// TIA Portal project "nalewak_v1" (V20)

(* hardware
DEVICE "S7-1500/ET200MP station_1"  S7-1500 station
   slot 0: "Rail_0"  Rack  6ES7 590-1***0-0AA0
   slot 1: "PLC_1"  CPU 1515-2 PN  6ES7 515-2AN03-0AB0  V3.1
      slot 3: "CPU display_1"  6ES7591-1BA00-0AA0
      slot 32768: "PROFINET interface_1"  X1
         slot 32769: "Port_1"  X1 P1
         slot 32770: "Port_2"  X1 P2
      slot 33024: "PROFINET interface_2"  X2
         slot 33025: "Port_1"  X2 P1
      slot 34817: "Virtual CP interface port_1"  Virtual CP interface port  Virtual CP interface port
   slot 2: "AI 8xHART HF_1"  AI 8xHART HF  6ES7 531-7TF00-0AB0  V1.0
   slot 3: "AQ 4xU/I HF_1"  AQ 4xU/I HF  6ES7 532-5ND00-0AB0  V1.1
   slot 4: "DI 32x24VDC BA_1"  DI 32x24VDC BA  6ES7 521-1BL10-0AA0  V1.1
   slot 5: "DQ 32x24VDC/0.5A BA_1"  DQ 32x24VDC/0.5A BA  6ES7 522-1BL10-0AA0  V1.1
DEVICE "PC-System_1"  SIMATIC PC station
   slot 0: "SIMATIC PC station"  Rail  SIMATIC PC-Station  V1.0
      slot 125: "Stationmanager"  Station_Manager  V6.0.4
   slot 1: "HMI_RT_1"  WinCC RT Advanced  6AV2 104-0xxxx-xxxx  17.0.0.0
      slot 33792: "Computer interface"  Host interface
   slot 2: "IE general_1"  IE General  IE_CP  V8.2.0
      slot 1: "PROFINET interface"  IEGeneral.Interface.8.2.0
*)

// ===== PLC "PLC_1"  CPU 1515-2 PN =====

VAR_GLOBAL   // PLC tag table "Default tag table"
   "System_Byte" AT %MB1 : Byte;
   "Clock_Byte" AT %MB0 : Byte;
   "Clock_10Hz" AT %M0.0 : Bool;
   "Clock_5Hz" AT %M0.1 : Bool;
   "Clock_2.5Hz" AT %M0.2 : Bool;
   "Clock_2Hz" AT %M0.3 : Bool;
   "Clock_1.25Hz" AT %M0.4 : Bool;
   "Clock_1Hz" AT %M0.5 : Bool;
   "Clock_0.625Hz" AT %M0.6 : Bool;
   "Clock_0.5Hz" AT %M0.7 : Bool;
   "Tag_1" AT %M4.3 : Bool;
   "porusz_cysterne" AT %M10.1 : Bool;
END_VAR

VAR_GLOBAL   // PLC tag table "PLC_tag"
   "ZS_001" AT %I16.0 : Bool;   // Czujnik przed wagą (wjazdowy)
   "ZS_002" AT %I16.1 : Bool;   // Czujnik za wagą (wyjazdowy)
   "PT1" AT %IW0 : Int;   // PT1 czujnik cisnienia1
   "PT2" AT %IW2 : Int;   // PT2 czujnik cisnienia2
   "PT3" AT %IW4 : Int;   // PT3 czujnik cisnienia3
   "PT4" AT %IW6 : Int;   // PT4 czujnik cisnienia4
   "TT1" AT %IW8 : Int;   // TT1 czujnik temperatury1
   "TT2" AT %IW10 : Int;   // TT2 czujnik temperatury2
   "TT3" AT %IW12 : Int;   // TT3 czujnik temperatury3
   "Waga" AT %IW14 : Int;   // MOST WAGI, waży cysterne z dokładnąćą +-10kg
   "FV_001" AT %QW0 : Int;   // Sterowanie zworem pierwszym
   "FV_002" AT %QW2 : Int;   // Sterowanie zworem drugim
   "U1" AT %Q8.1 : Bool;   // Uziemienie
   "LSHH_001" AT %I16.2 : Bool;   // Czujnik przelania (kamertonowy)
   "xv1.1" AT %Q8.2 : Bool;   // elektrozawór
   "xv1.2" AT %Q8.3 : Bool;   // elektrozawór
   "xv2.1" AT %Q8.4 : Bool;   // elektrozawór
   "xv2.2" AT %Q8.5 : Bool;   // elektrozawór
   "xv3.1" AT %Q8.6 : Bool;   // elektrozawór
   "xv3.2" AT %Q8.7 : Bool;   // elektrozawór
   "liczenie_prze2" AT %Q0.2 : Bool;   // Sygnał do licznika
   "M3" AT %Q8.0 : Bool;   // Zasilanie przciągarki M3~
END_VAR

VAR_GLOBAL   // PLC tag table "Var_tag"
   "Przycisk_Start" AT %M4.1 : Bool;   // Start
   "AWARIA" AT %M4.2 : Bool;   // Awaria
   "res3" AT %M10.3 : Bool;   // Zmienna pomocnicza
   "STOP" AT %M14.1 : Bool;
   "Brak_kolejnej_cysterny" AT %M14.3 : Bool;
   "Kolejna_cysterna" AT %M14.4 : Bool;
   "DRUKOWANIE" AT %M14.5 : Bool;   // drukowanie dokumentów
   "DRUK_END" AT %M14.6 : Bool;   // zakończenie drukowania dokumentów
   "ZEZ_1" AT %M14.7 : Bool;   // Zezwolenia na odjazd
   "ODJZD" AT %M15.0 : Bool;   // Odjazd
   "otw_zzaw1" AT %M15.1 : Bool;
   "otw_zzaw2" AT %M15.2 : Bool;
   "otw_zzaw3" AT %M15.3 : Bool;
   "TAR" AT %M20.3 : Bool;   // Przycisk na panelu hmi do tarowania
   "TAR2" AT %M20.5 : Bool;   // Przycisk na panelu hmi do tarowania
   "STR_NALEW" AT %M20.6 : Bool;   // Przycisk na panelu hmi start nalewu
   "POT_NALEW" AT %M20.7 : Bool;   // Potwierdzenie startu nalewu
   "dyspozycja_nalewy_start" AT %M21.0 : Bool;   // start nalewu
   "PROD1" AT %M21.1 : Bool;   // produkt1
   "pot_U1" AT %M21.2 : Bool;   // Potwierdzenie uziemienia
   "PROD2" AT %M21.3 : Bool;   // produkt2
   "PROD3" AT %M21.4 : Bool;   // produkt3
   "WART_ZAD" AT %M21.5 : Bool;   // wartość zadana została podana w panelu hmi
   "K_DYSPOZYCJI" AT %M21.6 : Bool;   // KONIEC DYSPOZYCJI
   "Opuszczona_rura" AT %M21.7 : Bool;   // Opuszczenie rury nalewczej
   "START_zestawienia" AT %M22.0 : Bool;   // Start zestawienia rur
   "Koniec_zestawienia_" AT %M22.1 : Bool;   // koniec zestawienia można przejść dalej
   "Zakonczenie_nalewu" AT %M22.2 : Bool;   // KOniec nalewu
   "Odzyskoop" AT %M22.3 : Bool;   // Odzysk oparów które unosząsie w cysternie
   "dddd" AT %MD24 : Real;
   "Zrzut_paliwa" AT %M28.0 : Bool;   // Oczyszcznie rury z resztek paliwa
END_VAR

TYPE "User_data_type_1"
   STRUCT
      Cos1 : Array[0..1] of Bool;
   END_STRUCT;
END_TYPE

DATA_BLOCK "Data_block_1"   // DB1
TITLE = Motor
{ S7_Optimized_Access := 'TRUE' }
VERSION : 0.1
BEGIN
END_DATA_BLOCK

DATA_BLOCK "nalewanie_DB_1"   // DB2
{ S7_Optimized_Access := 'TRUE' }
VERSION : 0.1
// stored: InstanceOfName nalewanie
"nalewanie"
BEGIN
END_DATA_BLOCK

DATA_BLOCK "Podstawienie cysterny kolejowej_DB"   // DB4
{ S7_Optimized_Access := 'TRUE' }
VERSION : 0.1
// stored: InstanceOfName Podstawienie cysterny kolejowej
"Podstawienie cysterny kolejowej"
BEGIN
END_DATA_BLOCK

DATA_BLOCK "nalewanie_DB"   // DB5
{ S7_Optimized_Access := 'TRUE' }
VERSION : 0.1
// stored: InstanceOfName nalewanie
"nalewanie"
BEGIN
END_DATA_BLOCK

DATA_BLOCK "Wstępne tarowanie cysterny kolejowej oraz weryfikacja, czy podstawiona cysterna kolejowa_DB_1"   // DB8
{ S7_Optimized_Access := 'TRUE' }
VERSION : 0.1
// stored: InstanceOfName Wstępne tarowanie cysterny kolejowej oraz weryfikacja, czy podstawiona cysterna kolejowa
"Wstępne tarowanie cysterny kolejowej oraz weryfikacja, czy podstawiona cysterna kolejowa"
BEGIN
END_DATA_BLOCK

DATA_BLOCK "Wstępne tarowanie cysterny kolejowej oraz weryfikacja, czy podstawiona cysterna kolejowa_DB"   // DB9
{ S7_Optimized_Access := 'TRUE' }
VERSION : 0.1
// stored: InstanceOfName Wstępne tarowanie cysterny kolejowej oraz weryfikacja, czy podstawiona cysterna kolejowa
"Wstępne tarowanie cysterny kolejowej oraz weryfikacja, czy podstawiona cysterna kolejowa"
BEGIN
END_DATA_BLOCK

DATA_BLOCK "przeciagarka2_DB_1"   // DB10
{ S7_Optimized_Access := 'TRUE' }
VERSION : 0.1
// stored: InstanceOfName przeciagarka2
"przeciagarka2"
BEGIN
END_DATA_BLOCK

DATA_BLOCK "przeciagarka2_DB"   // DB14
{ S7_Optimized_Access := 'TRUE' }
VERSION : 0.1
// stored: InstanceOfName przeciagarka2
"przeciagarka2"
BEGIN
END_DATA_BLOCK

DATA_BLOCK "Podstawienie cysterny kolejowej_DB_1"   // DB15
{ S7_Optimized_Access := 'TRUE' }
VERSION : 0.1
// stored: InstanceOfName Podstawienie cysterny kolejowej
"Podstawienie cysterny kolejowej"
BEGIN
END_DATA_BLOCK

DATA_BLOCK "Tarowanie_cysterny_kolejowej_DB_2"   // DB16
{ S7_Optimized_Access := 'TRUE' }
VERSION : 0.1
// stored: InstanceOfName Wstępne tarowanie cysterny kolejowej oraz weryfikacja, czy podstawiona cysterna kolejowa
"Wstępne tarowanie cysterny kolejowej oraz weryfikacja, czy podstawiona cysterna kolejowa"
BEGIN
END_DATA_BLOCK

DATA_BLOCK "Wstępne tarowanie cysterny kolejowej oraz weryfikacja, czy podstawiona cysterna kolejowa_DB_3"   // DB17
{ S7_Optimized_Access := 'TRUE' }
VERSION : 0.1
// stored: InstanceOfName Wstępne tarowanie cysterny kolejowej oraz weryfikacja, czy podstawiona cysterna kolejowa
"Wstępne tarowanie cysterny kolejowej oraz weryfikacja, czy podstawiona cysterna kolejowa"
BEGIN
END_DATA_BLOCK

DATA_BLOCK "Odpowietrzenie_rury_DB"   // DB19
{ S7_Optimized_Access := 'TRUE' }
VERSION : 0.1
// stored: InstanceOfName Odpowietrzenie_rury
"Odpowietrzenie_rury"
BEGIN
END_DATA_BLOCK

DATA_BLOCK "Parametry_Nalewania_DB"   // DB21
{ S7_Optimized_Access := 'TRUE' }
VERSION : 0.1
   VAR
      Waga_Paliwa_Zadana : Real;
   END_VAR
   VAR RETAIN
      Waga_Overshoot : Real;
      Czas_Zamykania_Zaworu : Real;
   END_VAR
   VAR
      Wymus_Miekki_Start : Bool;
      Wymus_Nalew_Dokladny : Bool;
      Waga_oczekiwana : Real;
      Waga_Punkt_Hamowania : Real;
      Wymus_Nalew_szybki : Bool;
      Waga_Zamykania : Bool;
   END_VAR
BEGIN
END_DATA_BLOCK

DATA_BLOCK "WAGA_do_PID_DB"   // DB24
{ S7_Optimized_Access := 'TRUE' }
VERSION : 0.1
   VAR
      WAGA_10s_temu : Real;   // Wartość "zamrożona" sprzed 10 sekund do obliczeń.
      Aktualna_Waga_Real : Real;   // Aktualna waga z mostu (już po skalowaniu na kg).
      Przeplyw_kg_s : Real;   // Wynikowy przepływ w tonach na godzinę.
      Waga_m1 : Real;   // Waga cysterny
      Waga_m2 : Real;   // Waga po dociśnięci nalewaka
      Waga_m3 : Real;   // Wartość zadana dla nelewu powolnego
      Waga_m4 : Real;   // Wartość zadana dla nelewu szybkiego
      Waga_m5 : Real;   // Wartość zadana dla nelewu dokładnego
      Waga_m6 : Real;   // Wartość zadan dla nalewu
      Waga_m6_1 : Real;   // Wartość zadan dla nalewu dokładnie policzona
      Waga_m7 : Real;   // Waga końcowa paliwa po wyjęciu lancy plus cysterna
      Waga_paliwa_zad : Real;   // Zadne ilość paliwa
      Waga_paliwa : Real;   // Końcowa waga paliwa
   END_VAR
BEGIN
END_DATA_BLOCK

DATA_BLOCK "Kalkulacja_wagi_na_tony/godzine_DB"   // DB28
{ S7_Optimized_Access := 'TRUE' }
VERSION : 0.1
// stored: InstanceOfName Kalkualcja
"Kalkualcja"
BEGIN
END_DATA_BLOCK

// folder: System blocks/Program resources

DATA_BLOCK "IEC_Timer_0_DB"   // DB11
{ S7_Optimized_Access := 'TRUE' }
AUTHOR : Simatic
FAMILY : IEC
NAME : IEC_TMR
VERSION : 1.0
// stored: InstanceOfName IEC_TIMER
"IEC_TIMER"
BEGIN
END_DATA_BLOCK

DATA_BLOCK "IEC_Counter_0_DB_3"   // DB12
{ S7_Optimized_Access := 'TRUE' }
AUTHOR : Simatic
FAMILY : IEC
NAME : CNTR
VERSION : 1.0
// stored: InstanceOfName IEC_COUNTER
"IEC_COUNTER"
BEGIN
END_DATA_BLOCK

DATA_BLOCK "IEC_Counter_0_DB_4"   // DB13
{ S7_Optimized_Access := 'TRUE' }
AUTHOR : Simatic
FAMILY : IEC
NAME : CNTR
VERSION : 1.0
// stored: InstanceOfName IEC_COUNTER
"IEC_COUNTER"
BEGIN
END_DATA_BLOCK

DATA_BLOCK "CZYSZCZENIE_RURY"   // DB18
{ S7_Optimized_Access := 'TRUE' }
AUTHOR : Simatic
FAMILY : IEC
NAME : IEC_TMR
VERSION : 1.0
// stored: InstanceOfName IEC_TIMER
"IEC_TIMER"
BEGIN
END_DATA_BLOCK

// folder: (top level)

FUNCTION_BLOCK "Wykrywanie przelania"   // FB1, LAD
{ S7_Optimized_Access := 'TRUE' }
VERSION : 0.1
BEGIN
END_FUNCTION_BLOCK

FUNCTION_BLOCK "3. Ustawienie dyspozycji nalewu (rodzaj produktu i jego ilość)"   // FB2, LAD
{ S7_Optimized_Access := 'TRUE' }
VERSION : 0.1
BEGIN
END_FUNCTION_BLOCK

FUNCTION_BLOCK "Podstawienie cysterny kolejowej"   // FB3, LAD
{ S7_Optimized_Access := 'TRUE' }
VERSION : 0.1
   VAR_OUTPUT
      cysterna_na_pozycji : Bool;
   END_VAR
BEGIN

REGION Network 1
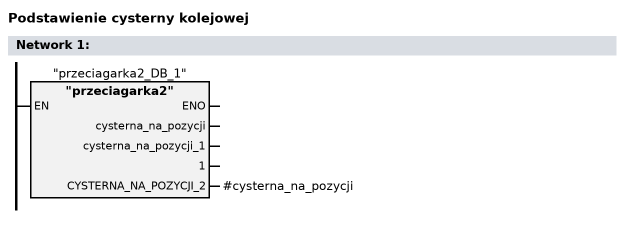
   RUNG wire#powerrail
      "przeciagarka2_DB_1"(cysterna_na_pozycji =>, cysterna_na_pozycji_1 =>, "1" =>, CYSTERNA_NA_POZYCJI_2 => #cysterna_na_pozycji)
   END_RUNG
   // the same network as SCL:
   "przeciagarka2_DB_1"(CYSTERNA_NA_POZYCJI_2 => #cysterna_na_pozycji);   // "przeciagarka2"
END_REGION
END_FUNCTION_BLOCK

FUNCTION_BLOCK "Wstępne tarowanie cysterny kolejowej oraz weryfikacja, czy podstawiona cysterna kolejowa"   // FB4, LAD
{ S7_Optimized_Access := 'TRUE' }
VERSION : 0.1
   VAR_INPUT
      tarow : Bool;   // start tarowanie
   END_VAR
   VAR_OUTPUT
      "2" : Bool;
   END_VAR
   VAR
      TON1 : IEC_TIMER;
   END_VAR
   VAR_TEMP
      "1" : Bool;
   END_VAR
BEGIN

REGION Network 1
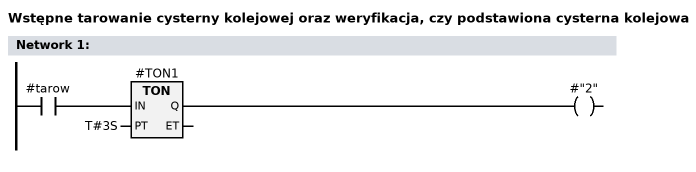
   #TON1.TON(IN := #tarow, PT := T#3S);
   #"2" := #TON1.Q;
END_REGION
END_FUNCTION_BLOCK

FUNCTION_BLOCK "nalewanie"   // FB5, LAD
{ S7_Optimized_Access := 'TRUE' }
VERSION : 0.1
   VAR_OUTPUT
      koniec_etapu_nalewania : Bool;
   END_VAR
   VAR
      ton : IEC_TIMER;
      Flow_ref_ms : Real := 70.0;   // Miekki_Start wartość dla niego w [kg/s]
      Flow_ref_ns : Real := 175.0;   // Nalew_szybki wartość dla niego w [kg/s]
      Flow_ref_Nd : Real := 43.75;   // Nalew_Dokladny wartość dla niego w [kg/s]
   END_VAR
   VAR_TEMP
      Cel_Dla_PID : Real;
      Waga_Znormalizowana : Real;
      Procent_Z_PID : Real;
      Sygnal_Analogowy_Int : Int;
      Zawor_W_Procentach : Real;
      ramp_out : Real;
      Wartość_dla_PID : Real;
   END_VAR
BEGIN

REGION Network 1
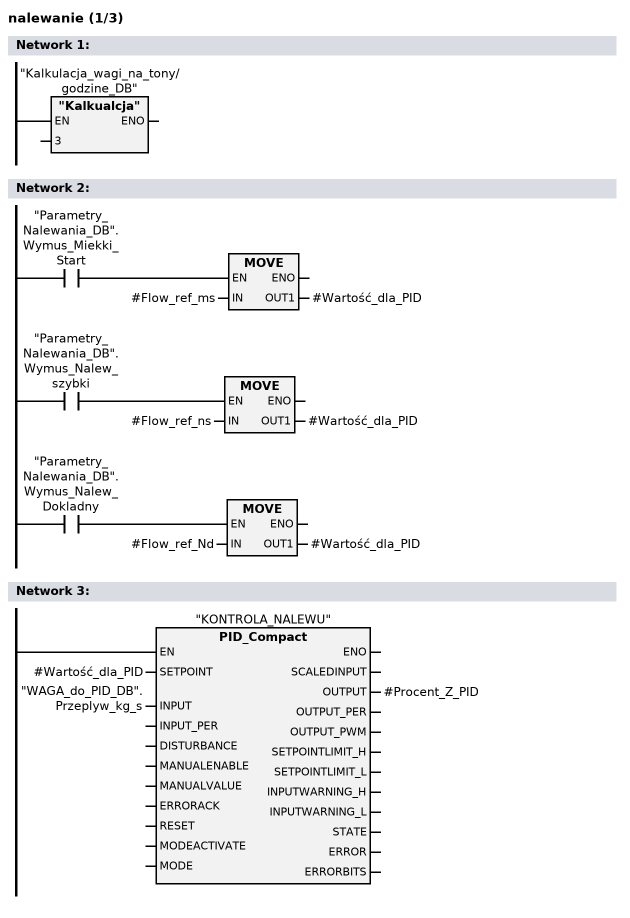
   RUNG wire#powerrail
      "Kalkulacja_wagi_na_tony/godzine_DB"("3" :=)
   END_RUNG
   // the same network as SCL:
   "Kalkulacja_wagi_na_tony/godzine_DB"();   // "Kalkualcja"
END_REGION

REGION Network 2
   RUNG wire#powerrail
      Contact( "Parametry_Nalewania_DB".Wymus_Miekki_Start )
      Move(in := #Flow_ref_ms, out1 => #Wartość_dla_PID)
   END_RUNG
   RUNG wire#powerrail
      Contact( "Parametry_Nalewania_DB".Wymus_Nalew_szybki )
      Move(in := #Flow_ref_ns, out1 => #Wartość_dla_PID)
   END_RUNG
   RUNG wire#powerrail
      Contact( "Parametry_Nalewania_DB".Wymus_Nalew_Dokladny )
      Move(in := #Flow_ref_Nd, out1 => #Wartość_dla_PID)
   END_RUNG
   // the same network as SCL:
   IF "Parametry_Nalewania_DB".Wymus_Miekki_Start THEN #Wartość_dla_PID := #Flow_ref_ms; END_IF;
   IF "Parametry_Nalewania_DB".Wymus_Nalew_szybki THEN #Wartość_dla_PID := #Flow_ref_ns; END_IF;
   IF "Parametry_Nalewania_DB".Wymus_Nalew_Dokladny THEN #Wartość_dla_PID := #Flow_ref_Nd; END_IF;
END_REGION

REGION Network 3
   "KONTROLA_NALEWU"(Setpoint := #Wartość_dla_PID,   // PID_Compact
                     Input := "WAGA_do_PID_DB".Przeplyw_kg_s,
                     Output => #Procent_Z_PID);
END_REGION

REGION Network 4
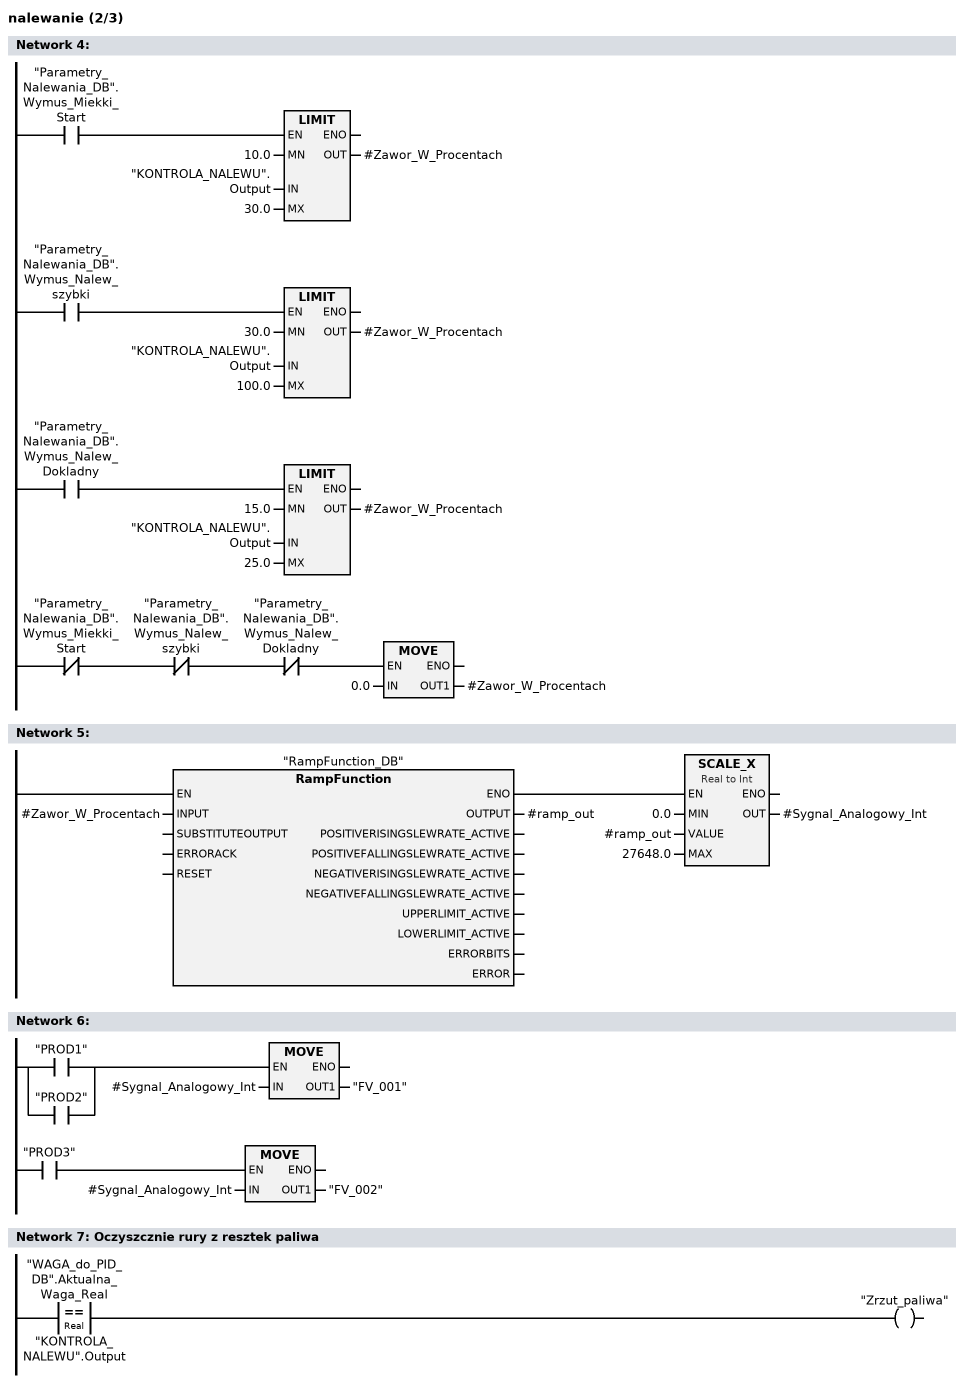
   IF "Parametry_Nalewania_DB".Wymus_Miekki_Start THEN
       #Zawor_W_Procentach := LIMIT(MN := 10.0, IN := "KONTROLA_NALEWU".Output, MX := 30.0);
   END_IF;
   IF "Parametry_Nalewania_DB".Wymus_Nalew_szybki THEN
       #Zawor_W_Procentach := LIMIT(MN := 30.0, IN := "KONTROLA_NALEWU".Output, MX := 100.0);
   END_IF;
   IF "Parametry_Nalewania_DB".Wymus_Nalew_Dokladny THEN
       #Zawor_W_Procentach := LIMIT(MN := 15.0, IN := "KONTROLA_NALEWU".Output, MX := 25.0);
   END_IF;
   IF NOT "Parametry_Nalewania_DB".Wymus_Miekki_Start AND NOT "Parametry_Nalewania_DB".Wymus_Nalew_szybki AND NOT "Parametry_Nalewania_DB".Wymus_Nalew_Dokladny THEN
       #Zawor_W_Procentach := 0.0;
   END_IF;
END_REGION

REGION Network 5
   // ENO of a box is taken as its EN; it also drops when the box reports an error
   "RampFunction_DB"(Input := #Zawor_W_Procentach, Output => #ramp_out);   // RampFunction
   #Sygnal_Analogowy_Int := SCALE_X(MIN := 0.0, VALUE := #ramp_out, MAX := 27648.0);
END_REGION

REGION Network 6
   RUNG wire#powerrail
      Contact( "PROD1" )
      wire#w1
      Move(in := #Sygnal_Analogowy_Int, out1 => "FV_001")
   END_RUNG
   RUNG wire#powerrail
      Contact( "PROD2" )
   END_RUNG wire#w1
   RUNG wire#powerrail
      Contact( "PROD3" )
      Move(in := #Sygnal_Analogowy_Int, out1 => "FV_002")
   END_RUNG
   // the same network as SCL:
   IF "PROD1" OR "PROD2" THEN "FV_001" := #Sygnal_Analogowy_Int; END_IF;
   IF "PROD3" THEN "FV_002" := #Sygnal_Analogowy_Int; END_IF;
END_REGION

REGION Network 7: Oczyszcznie rury z resztek paliwa
   RUNG wire#powerrail
      { S7_Templates := "SrcType := Real" } EQ_Contact(in1 := "WAGA_do_PID_DB".Aktualna_Waga_Real, in2 := "KONTROLA_NALEWU".Output)
      Coil( "Zrzut_paliwa" )
   END_RUNG
   // the same network as SCL:
   "Zrzut_paliwa" := "WAGA_do_PID_DB".Aktualna_Waga_Real = "KONTROLA_NALEWU".Output;
END_REGION

REGION Network 8: Oczyszcznie rury z resztek paliwa
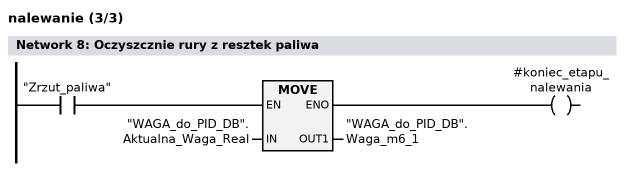
   RUNG wire#powerrail
      Contact( "Zrzut_paliwa" )
      Move(in := "WAGA_do_PID_DB".Aktualna_Waga_Real, out1 => "WAGA_do_PID_DB".Waga_m6_1)
      Coil( #koniec_etapu_nalewania )
   END_RUNG
   // the same network as SCL:
   IF "Zrzut_paliwa" THEN "WAGA_do_PID_DB".Waga_m6_1 := "WAGA_do_PID_DB".Aktualna_Waga_Real; END_IF;
   #koniec_etapu_nalewania := "Zrzut_paliwa";
END_REGION
END_FUNCTION_BLOCK

FUNCTION_BLOCK "przeciagarka2"   // FB6, LAD
{ S7_Optimized_Access := 'TRUE' }
VERSION : 0.1
   VAR_OUTPUT
      cysterna_na_pozycji : Bool;
      cysterna_na_pozycji_1 : Bool;
      "1" : Bool;
      CYSTERNA_NA_POZYCJI_2 : Bool;
   END_VAR
   VAR
      reset1 : Bool;
      reset2 : Bool;
      Kolejna_cysterna : Bool;
      pamieczbocz_3 : Bool;
      pamieczbocz_1 : Bool;
      pamieczbocz_2 : Bool;
   END_VAR
   VAR_TEMP   // added for the SCL form of the ladder/FBD networks
      _w1 : Bool;
   END_VAR
BEGIN

REGION Network 1: Zasilanie przciągarki M3~
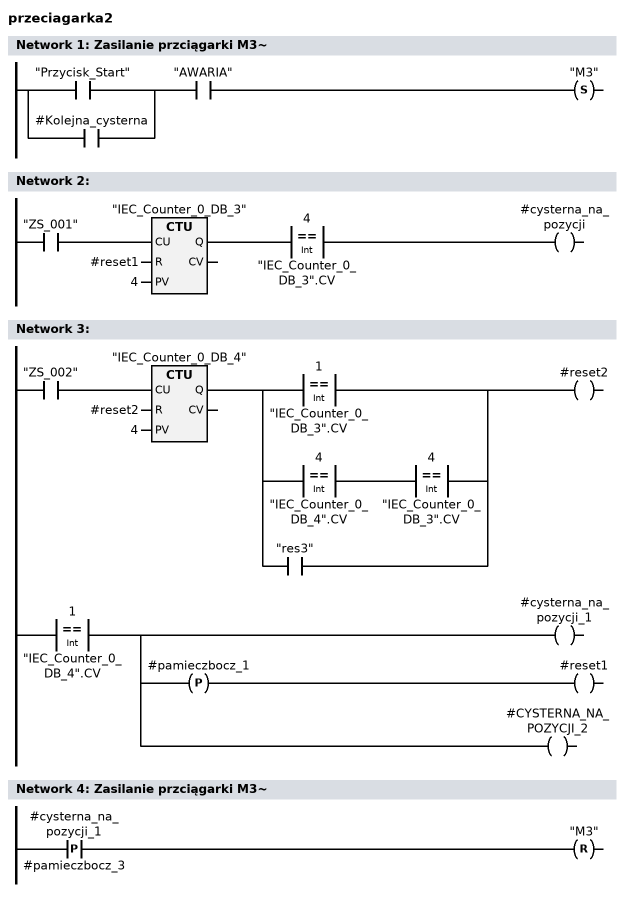
   RUNG wire#powerrail
      Contact( "Przycisk_Start" )
      wire#w1
      Contact( "AWARIA" )
      S_Coil( "M3" )
   END_RUNG
   RUNG wire#powerrail
      Contact( #Kolejna_cysterna )
   END_RUNG wire#w1
   // the same network as SCL:
   IF ("Przycisk_Start" OR #Kolejna_cysterna) AND "AWARIA" THEN "M3" := TRUE; END_IF;
END_REGION

REGION Network 2
   "IEC_Counter_0_DB_3".CTU(CU := "ZS_001", R := #reset1, PV := 4);
   #cysterna_na_pozycji := "IEC_Counter_0_DB_3".Q AND (4 = "IEC_Counter_0_DB_3".CV);
END_REGION

REGION Network 3
   "IEC_Counter_0_DB_4".CTU(CU := "ZS_002", R := #reset2, PV := 4);
   #reset2 := "IEC_Counter_0_DB_4".Q AND ((1 = "IEC_Counter_0_DB_3".CV) OR ((4 = "IEC_Counter_0_DB_4".CV) AND (4 = "IEC_Counter_0_DB_3".CV)) OR "res3");
   #cysterna_na_pozycji_1 := 1 = "IEC_Counter_0_DB_4".CV;
   #_w1 := #cysterna_na_pozycji_1 AND NOT #pamieczbocz_1;   // rising edge
   #pamieczbocz_1 := #cysterna_na_pozycji_1;
   #reset1 := #_w1;
   #CYSTERNA_NA_POZYCJI_2 := #cysterna_na_pozycji_1;
END_REGION

REGION Network 4: Zasilanie przciągarki M3~
   RUNG wire#powerrail
      P_Contact(operand := #cysterna_na_pozycji_1, bit := #pamieczbocz_3)
      R_Coil( "M3" )
   END_RUNG
   // the same network as SCL:
   #_w1 := #cysterna_na_pozycji_1 AND NOT #pamieczbocz_3;   // rising edge of #cysterna_na_pozycji_1
   #pamieczbocz_3 := #cysterna_na_pozycji_1;
   IF #_w1 THEN "M3" := FALSE; END_IF;
END_REGION
END_FUNCTION_BLOCK

FUNCTION_BLOCK "Odpowietrzenie_rury"   // FB7, LAD
{ S7_Optimized_Access := 'TRUE' }
VERSION : 0.1
   VAR_INPUT
      odpowietrznie : Bool;   // wyrzuca resztki paliwa z rury po zamknięci zaworu
   END_VAR
   VAR_OUTPUT
      odpowietrznie_koniec : Bool;
   END_VAR
BEGIN

REGION Network 1
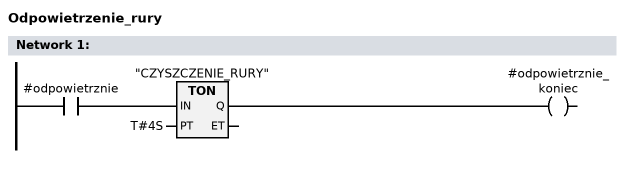
   "CZYSZCZENIE_RURY".TON(IN := #odpowietrznie, PT := T#4S);
   #odpowietrznie_koniec := "CZYSZCZENIE_RURY".Q;
END_REGION
END_FUNCTION_BLOCK

FUNCTION_BLOCK "Block_1"   // FB8, LAD
{ S7_Optimized_Access := 'TRUE' }
VERSION : 0.1
   VAR_OUTPUT
      "Koniec Nalewu" : Bool;
      "Następna cysterna" : Bool;
   END_VAR
BEGIN

REGION Network 1
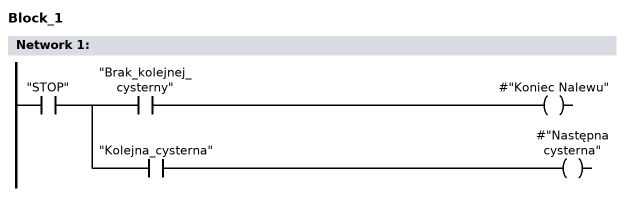
   RUNG wire#powerrail
      Contact( "STOP" )
      wire#w1
      Contact( "Brak_kolejnej_cysterny" )
      Coil( #"Koniec Nalewu" )
   END_RUNG
   RUNG wire#w1
      Contact( "Kolejna_cysterna" )
      Coil( #"Następna cysterna" )
   END_RUNG
   // the same network as SCL:
   #"Koniec Nalewu" := "STOP" AND "Brak_kolejnej_cysterny";
   #"Następna cysterna" := "STOP" AND "Kolejna_cysterna";
END_REGION
END_FUNCTION_BLOCK

FUNCTION_BLOCK "Kalkualcja"   // FB9, LAD
{ S7_Optimized_Access := 'TRUE' }
VERSION : 0.1
   VAR_INPUT
      "3" : Bool;
   END_VAR
   VAR_TEMP
      Zawor_W_Procentach : Real;
      Sygnal_Analogowy_Int : Int;
      "1" : Bool;
      wynik : Real;
      impuls : Bool;
      Zapas_Hamowania_kg : Real;
   END_VAR
BEGIN

REGION Network 1
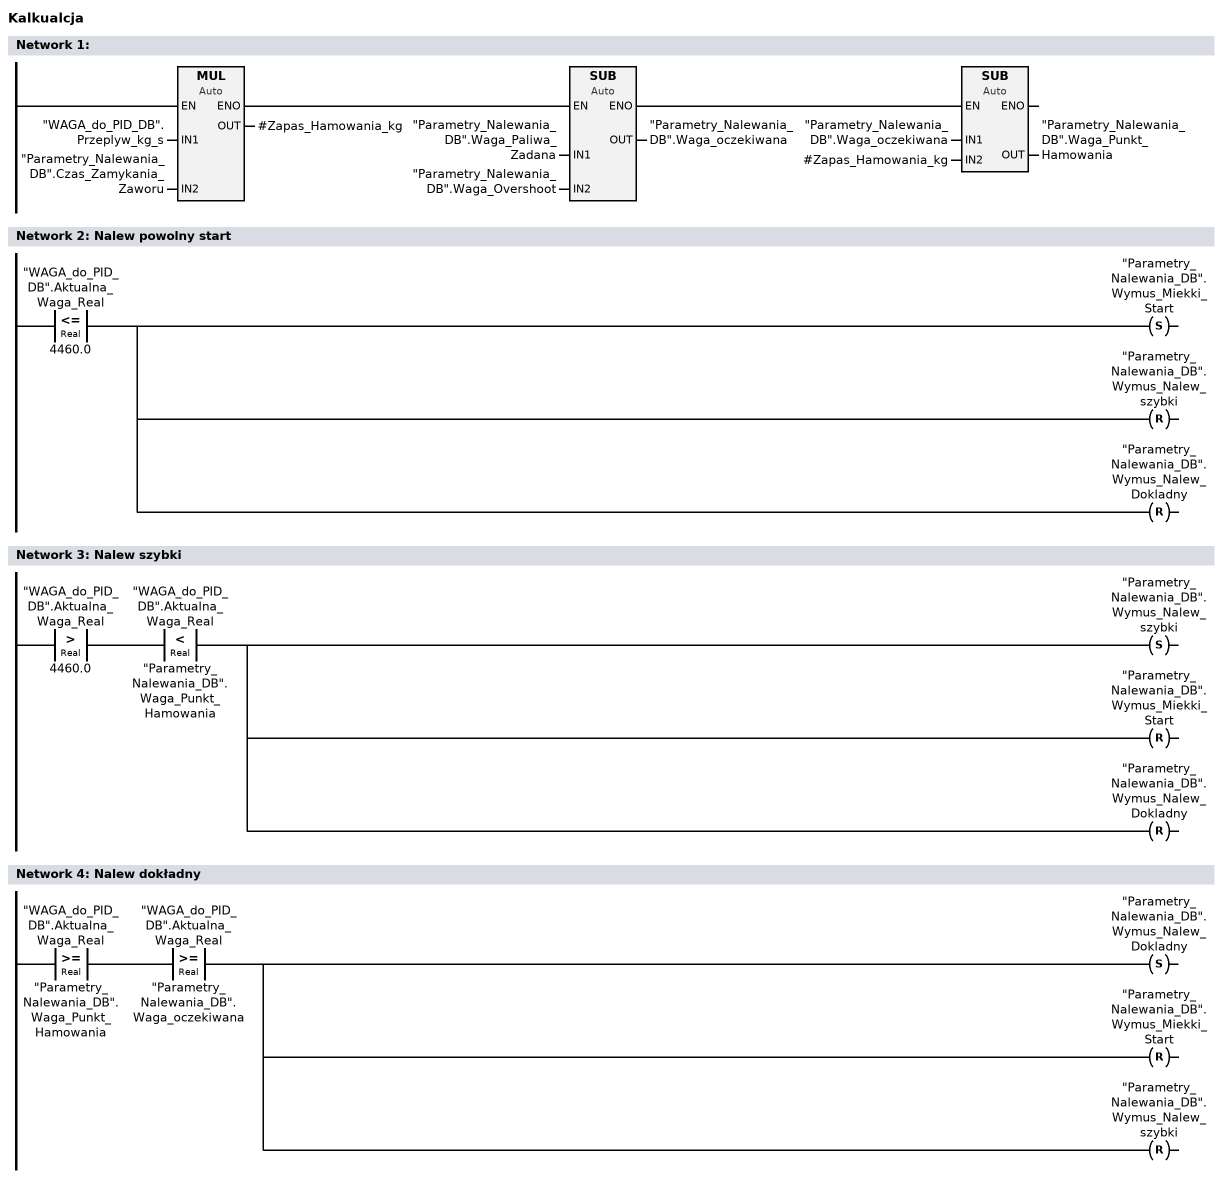
   RUNG wire#powerrail
      Mul(in1 := "WAGA_do_PID_DB".Przeplyw_kg_s, in2 := "Parametry_Nalewania_DB".Czas_Zamykania_Zaworu, out => #Zapas_Hamowania_kg)
      Sub(in1 := "Parametry_Nalewania_DB".Waga_Paliwa_Zadana, in2 := "Parametry_Nalewania_DB".Waga_Overshoot, out => "Parametry_Nalewania_DB".Waga_oczekiwana)
      Sub(in1 := "Parametry_Nalewania_DB".Waga_oczekiwana, in2 := #Zapas_Hamowania_kg, out => "Parametry_Nalewania_DB".Waga_Punkt_Hamowania)
   END_RUNG
   // the same network as SCL:
   #Zapas_Hamowania_kg := "WAGA_do_PID_DB".Przeplyw_kg_s * "Parametry_Nalewania_DB".Czas_Zamykania_Zaworu;
   "Parametry_Nalewania_DB".Waga_oczekiwana := "Parametry_Nalewania_DB".Waga_Paliwa_Zadana - "Parametry_Nalewania_DB".Waga_Overshoot;
   "Parametry_Nalewania_DB".Waga_Punkt_Hamowania := "Parametry_Nalewania_DB".Waga_oczekiwana - #Zapas_Hamowania_kg;
END_REGION

REGION Network 2: Nalew powolny start
   RUNG wire#powerrail
      { S7_Templates := "SrcType := Real" } LE_Contact(in1 := "WAGA_do_PID_DB".Aktualna_Waga_Real, in2 := 4460.0)
      wire#w1
      S_Coil( "Parametry_Nalewania_DB".Wymus_Miekki_Start )
   END_RUNG
   RUNG wire#w1
      R_Coil( "Parametry_Nalewania_DB".Wymus_Nalew_szybki )
   END_RUNG
   RUNG wire#w1
      R_Coil( "Parametry_Nalewania_DB".Wymus_Nalew_Dokladny )
   END_RUNG
   // the same network as SCL:
   IF "WAGA_do_PID_DB".Aktualna_Waga_Real <= 4460.0 THEN
       "Parametry_Nalewania_DB".Wymus_Miekki_Start := TRUE;
       "Parametry_Nalewania_DB".Wymus_Nalew_szybki := FALSE;
       "Parametry_Nalewania_DB".Wymus_Nalew_Dokladny := FALSE;
   END_IF;
END_REGION

REGION Network 3: Nalew szybki
   RUNG wire#powerrail
      { S7_Templates := "SrcType := Real" } GT_Contact(in1 := "WAGA_do_PID_DB".Aktualna_Waga_Real, in2 := 4460.0)
      { S7_Templates := "SrcType := Real" } LT_Contact(in1 := "WAGA_do_PID_DB".Aktualna_Waga_Real, in2 := "Parametry_Nalewania_DB".Waga_Punkt_Hamowania)
      wire#w1
      S_Coil( "Parametry_Nalewania_DB".Wymus_Nalew_szybki )
   END_RUNG
   RUNG wire#w1
      R_Coil( "Parametry_Nalewania_DB".Wymus_Miekki_Start )
   END_RUNG
   RUNG wire#w1
      R_Coil( "Parametry_Nalewania_DB".Wymus_Nalew_Dokladny )
   END_RUNG
   // the same network as SCL:
   IF ("WAGA_do_PID_DB".Aktualna_Waga_Real > 4460.0) AND ("WAGA_do_PID_DB".Aktualna_Waga_Real < "Parametry_Nalewania_DB".Waga_Punkt_Hamowania) THEN
       "Parametry_Nalewania_DB".Wymus_Nalew_szybki := TRUE;
       "Parametry_Nalewania_DB".Wymus_Miekki_Start := FALSE;
       "Parametry_Nalewania_DB".Wymus_Nalew_Dokladny := FALSE;
   END_IF;
END_REGION

REGION Network 4: Nalew dokładny
   RUNG wire#powerrail
      { S7_Templates := "SrcType := Real" } GE_Contact(in1 := "WAGA_do_PID_DB".Aktualna_Waga_Real, in2 := "Parametry_Nalewania_DB".Waga_Punkt_Hamowania)
      { S7_Templates := "SrcType := Real" } GE_Contact(in1 := "WAGA_do_PID_DB".Aktualna_Waga_Real, in2 := "Parametry_Nalewania_DB".Waga_oczekiwana)
      wire#w1
      S_Coil( "Parametry_Nalewania_DB".Wymus_Nalew_Dokladny )
   END_RUNG
   RUNG wire#w1
      R_Coil( "Parametry_Nalewania_DB".Wymus_Miekki_Start )
   END_RUNG
   RUNG wire#w1
      R_Coil( "Parametry_Nalewania_DB".Wymus_Nalew_szybki )
   END_RUNG
   // the same network as SCL:
   IF ("WAGA_do_PID_DB".Aktualna_Waga_Real >= "Parametry_Nalewania_DB".Waga_Punkt_Hamowania) AND ("WAGA_do_PID_DB".Aktualna_Waga_Real >= "Parametry_Nalewania_DB".Waga_oczekiwana) THEN
       "Parametry_Nalewania_DB".Wymus_Nalew_Dokladny := TRUE;
       "Parametry_Nalewania_DB".Wymus_Miekki_Start := FALSE;
       "Parametry_Nalewania_DB".Wymus_Nalew_szybki := FALSE;
   END_IF;
END_REGION
END_FUNCTION_BLOCK

ORGANIZATION_BLOCK "Main"   // OB1, LAD, ProgramCycle
TITLE = Nalewak
{ S7_Optimized_Access := 'TRUE' }
VERSION : 0.1
   VAR_INPUT
      Initial_Call : Bool;   // Initial call of this OB
      Remanence : Bool;   // =True, if remanent data are available
   END_VAR
   VAR_TEMP
      waf : Bool;
   END_VAR
   VAR_TEMP   // added for the SCL form of the ladder/FBD networks
      _w1 : Bool;
   END_VAR
BEGIN

REGION Network 1: Podstawienie cysterny
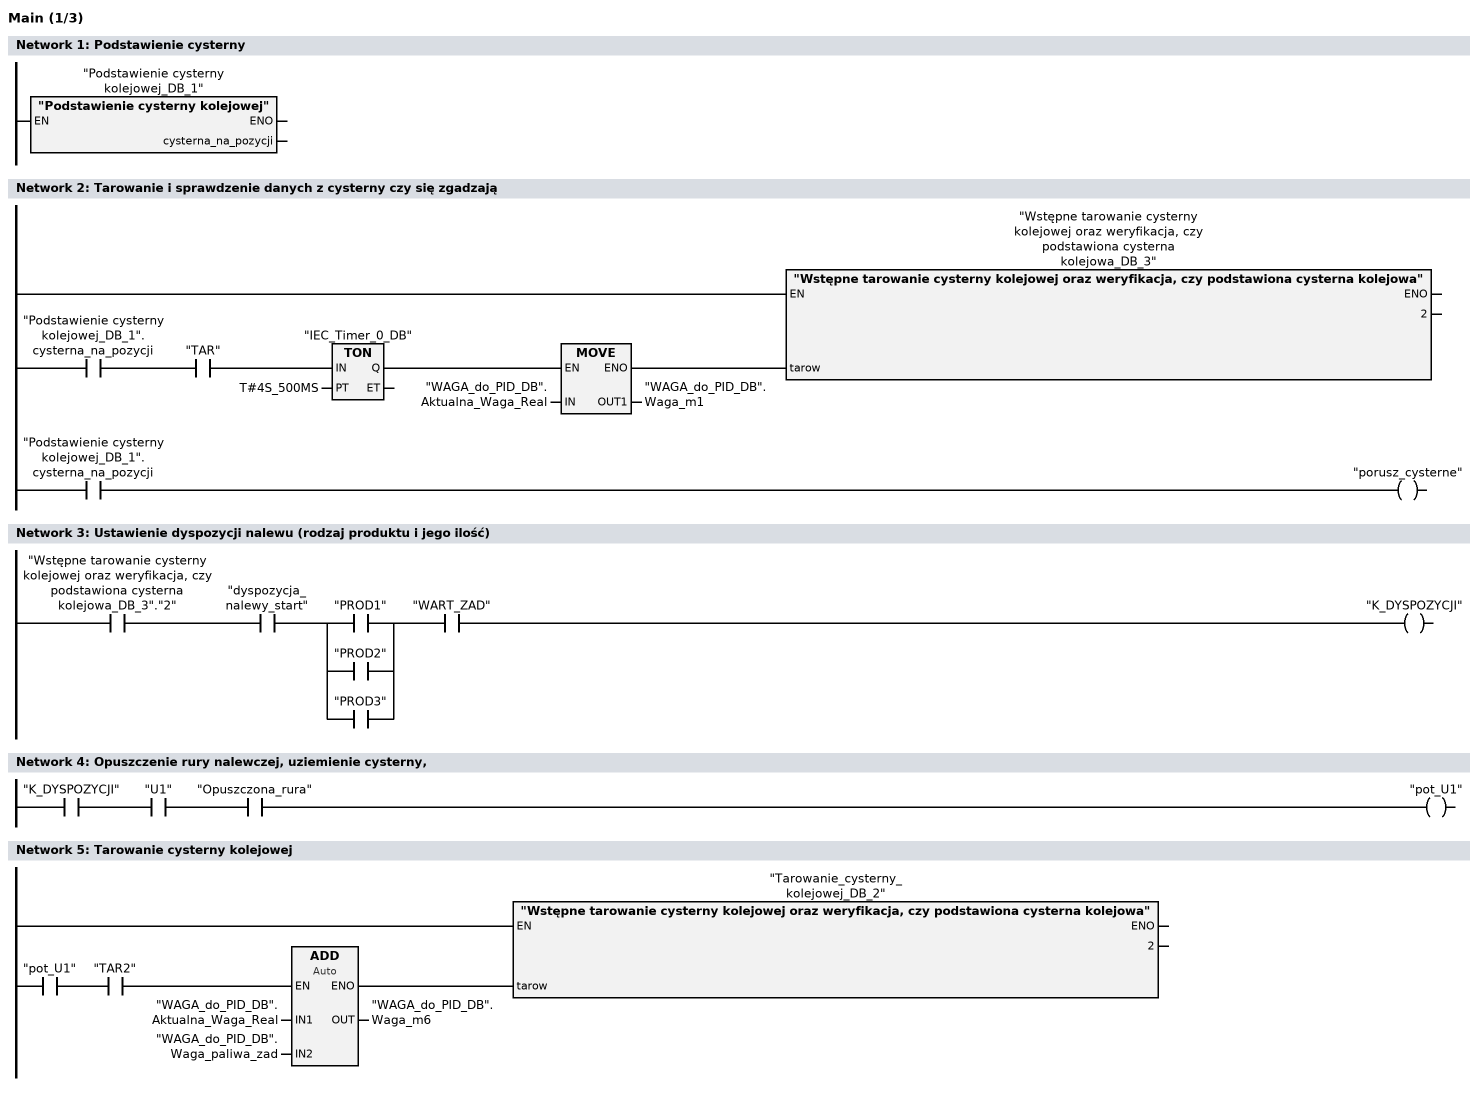
   RUNG wire#powerrail
      "Podstawienie cysterny kolejowej_DB_1"(cysterna_na_pozycji =>)
   END_RUNG
   // the same network as SCL:
   "Podstawienie cysterny kolejowej_DB_1"();   // "Podstawienie cysterny kolejowej"
END_REGION

REGION Network 2: Tarowanie i sprawdzenie danych z cysterny czy się zgadzają
   "IEC_Timer_0_DB".TON(IN := "Podstawienie cysterny kolejowej_DB_1".cysterna_na_pozycji AND "TAR",
                        PT := T#4S_500MS);
   IF "IEC_Timer_0_DB".Q THEN "WAGA_do_PID_DB".Waga_m1 := "WAGA_do_PID_DB".Aktualna_Waga_Real; END_IF;
   "Wstępne tarowanie cysterny kolejowej oraz weryfikacja, czy podstawiona cysterna kolejowa_DB_3"(tarow := "IEC_Timer_0_DB".Q);   // "Wstępne tarowanie cysterny kolejowej oraz weryfikacja, czy podstawiona cysterna kolejowa"
   "porusz_cysterne" := "Podstawienie cysterny kolejowej_DB_1".cysterna_na_pozycji;
END_REGION

REGION Network 3: Ustawienie dyspozycji nalewu (rodzaj produktu i jego ilość)
   RUNG wire#powerrail
      Contact( "Wstępne tarowanie cysterny kolejowej oraz weryfikacja, czy podstawiona cysterna kolejowa_DB_3"."2" )
      Contact( "dyspozycja_nalewy_start" )
      wire#w1
      Contact( "PROD1" )
      wire#w2
      Contact( "WART_ZAD" )
      Coil( "K_DYSPOZYCJI" )
   END_RUNG
   RUNG wire#w1
      Contact( "PROD2" )
   END_RUNG wire#w2
   RUNG wire#w1
      Contact( "PROD3" )
   END_RUNG wire#w2
   // the same network as SCL:
   "K_DYSPOZYCJI" := "Wstępne tarowanie cysterny kolejowej oraz weryfikacja, czy podstawiona cysterna kolejowa_DB_3"."2" AND "dyspozycja_nalewy_start" AND ("PROD1" OR "PROD2" OR "PROD3") AND "WART_ZAD";
END_REGION

REGION Network 4: Opuszczenie rury nalewczej, uziemienie cysterny,
   RUNG wire#powerrail
      Contact( "K_DYSPOZYCJI" )
      Contact( "U1" )
      Contact( "Opuszczona_rura" )
      Coil( "pot_U1" )
   END_RUNG
   // the same network as SCL:
   "pot_U1" := "K_DYSPOZYCJI" AND "U1" AND "Opuszczona_rura";
END_REGION

REGION Network 5: Tarowanie cysterny kolejowej
   RUNG wire#powerrail
      "Tarowanie_cysterny_kolejowej_DB_2"(tarow := wire#w1, "2" =>)
   END_RUNG
   RUNG wire#powerrail
      Contact( "pot_U1" )
      Contact( "TAR2" )
      Add(in1 := "WAGA_do_PID_DB".Aktualna_Waga_Real, in2 := "WAGA_do_PID_DB".Waga_paliwa_zad, out => "WAGA_do_PID_DB".Waga_m6)
   END_RUNG wire#w1
   // the same network as SCL:
   #_w1 := "pot_U1" AND "TAR2";
   IF #_w1 THEN
       "WAGA_do_PID_DB".Waga_m6 := "WAGA_do_PID_DB".Aktualna_Waga_Real + "WAGA_do_PID_DB".Waga_paliwa_zad;
   END_IF;
   "Tarowanie_cysterny_kolejowej_DB_2"(tarow := #_w1);   // "Wstępne tarowanie cysterny kolejowej oraz weryfikacja, czy podstawiona cysterna kolejowa"
END_REGION

REGION Network 6: Zestawienie trasy nalewu przez otwarcie/zamknięcie zaworów produktowych
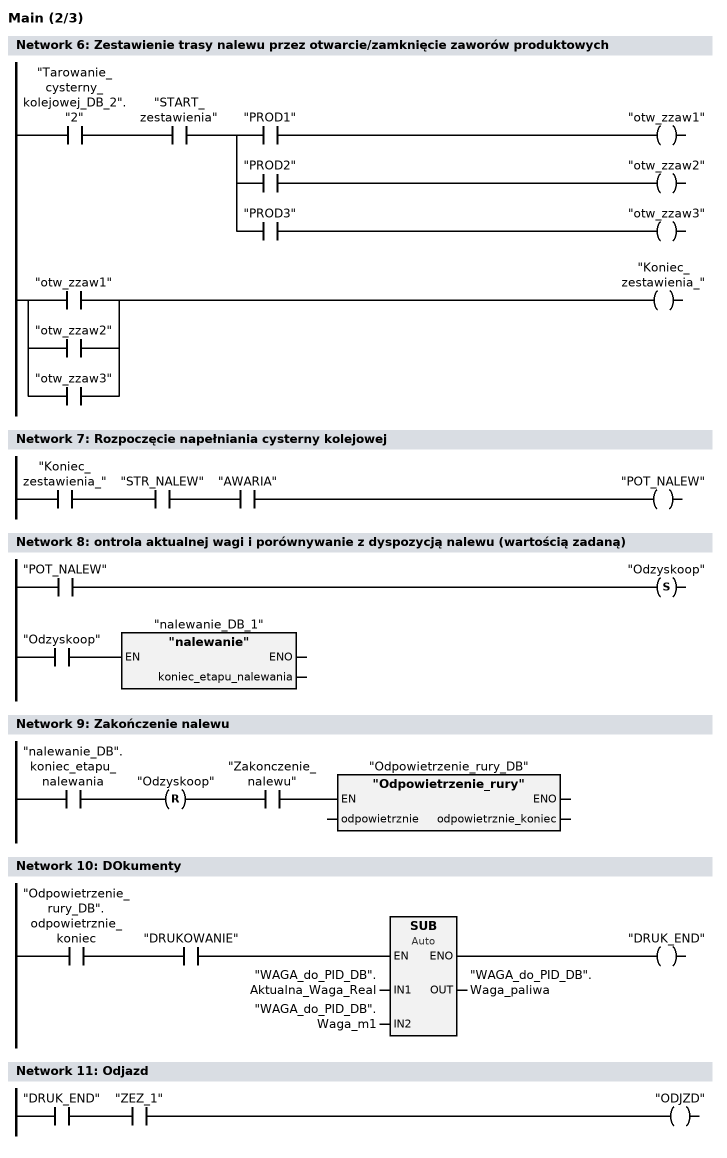
   RUNG wire#powerrail
      Contact( "Tarowanie_cysterny_kolejowej_DB_2"."2" )
      Contact( "START_zestawienia" )
      wire#w1
      Contact( "PROD1" )
      Coil( "otw_zzaw1" )
   END_RUNG
   RUNG wire#w1
      Contact( "PROD2" )
      Coil( "otw_zzaw2" )
   END_RUNG
   RUNG wire#w1
      Contact( "PROD3" )
      Coil( "otw_zzaw3" )
   END_RUNG
   RUNG wire#powerrail
      Contact( "otw_zzaw1" )
      wire#w2
      Coil( "Koniec_zestawienia_" )
   END_RUNG
   RUNG wire#powerrail
      Contact( "otw_zzaw2" )
   END_RUNG wire#w2
   RUNG wire#powerrail
      Contact( "otw_zzaw3" )
   END_RUNG wire#w2
   // the same network as SCL:
   #_w1 := "Tarowanie_cysterny_kolejowej_DB_2"."2" AND "START_zestawienia";
   "otw_zzaw1" := #_w1 AND "PROD1";
   "otw_zzaw2" := #_w1 AND "PROD2";
   "otw_zzaw3" := #_w1 AND "PROD3";
   "Koniec_zestawienia_" := "otw_zzaw1" OR "otw_zzaw2" OR "otw_zzaw3";
END_REGION

REGION Network 7: Rozpoczęcie napełniania cysterny kolejowej
   RUNG wire#powerrail
      Contact( "Koniec_zestawienia_" )
      Contact( "STR_NALEW" )
      Contact( "AWARIA" )
      Coil( "POT_NALEW" )
   END_RUNG
   // the same network as SCL:
   "POT_NALEW" := "Koniec_zestawienia_" AND "STR_NALEW" AND "AWARIA";
END_REGION

REGION Network 8: ontrola aktualnej wagi i porównywanie z dyspozycją nalewu (wartością zadaną)
   RUNG wire#powerrail
      Contact( "POT_NALEW" )
      S_Coil( "Odzyskoop" )
   END_RUNG
   RUNG wire#powerrail
      Contact( "Odzyskoop" )
      "nalewanie_DB_1"(koniec_etapu_nalewania =>)
   END_RUNG
   // the same network as SCL:
   IF "POT_NALEW" THEN "Odzyskoop" := TRUE; END_IF;
   IF "Odzyskoop" THEN
       "nalewanie_DB_1"();   // "nalewanie"
   END_IF;
END_REGION

REGION Network 9: Zakończenie nalewu
   RUNG wire#powerrail
      Contact( "nalewanie_DB".koniec_etapu_nalewania )
      R_Coil( "Odzyskoop" )
      Contact( "Zakonczenie_nalewu" )
      "Odpowietrzenie_rury_DB"(odpowietrznie :=, odpowietrznie_koniec =>)
   END_RUNG
   // the same network as SCL:
   IF "nalewanie_DB".koniec_etapu_nalewania THEN "Odzyskoop" := FALSE; END_IF;
   IF "nalewanie_DB".koniec_etapu_nalewania AND "Zakonczenie_nalewu" THEN
       "Odpowietrzenie_rury_DB"();   // "Odpowietrzenie_rury"
   END_IF;
END_REGION

REGION Network 10: DOkumenty
   RUNG wire#powerrail
      Contact( "Odpowietrzenie_rury_DB".odpowietrznie_koniec )
      Contact( "DRUKOWANIE" )
      Sub(in1 := "WAGA_do_PID_DB".Aktualna_Waga_Real, in2 := "WAGA_do_PID_DB".Waga_m1, out => "WAGA_do_PID_DB".Waga_paliwa)
      Coil( "DRUK_END" )
   END_RUNG
   // the same network as SCL:
   #_w1 := "Odpowietrzenie_rury_DB".odpowietrznie_koniec AND "DRUKOWANIE";
   IF #_w1 THEN
       "WAGA_do_PID_DB".Waga_paliwa := "WAGA_do_PID_DB".Aktualna_Waga_Real - "WAGA_do_PID_DB".Waga_m1;
   END_IF;
   "DRUK_END" := #_w1;
END_REGION

REGION Network 11: Odjazd
   RUNG wire#powerrail
      Contact( "DRUK_END" )
      Contact( "ZEZ_1" )
      Coil( "ODJZD" )
   END_RUNG
   // the same network as SCL:
   "ODJZD" := "DRUK_END" AND "ZEZ_1";
END_REGION

REGION Network 12: Blok techniczny
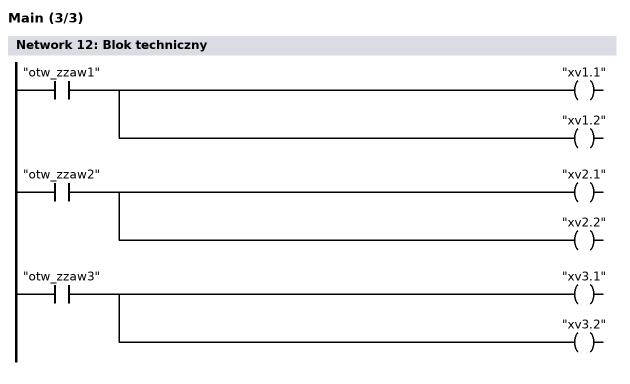
   RUNG wire#powerrail
      Contact( "otw_zzaw1" )
      wire#w1
      Coil( "xv1.1" )
   END_RUNG
   RUNG wire#w1
      Coil( "xv1.2" )
   END_RUNG
   RUNG wire#powerrail
      Contact( "otw_zzaw2" )
      wire#w2
      Coil( "xv2.1" )
   END_RUNG
   RUNG wire#w2
      Coil( "xv2.2" )
   END_RUNG
   RUNG wire#powerrail
      Contact( "otw_zzaw3" )
      wire#w3
      Coil( "xv3.1" )
   END_RUNG
   RUNG wire#w3
      Coil( "xv3.2" )
   END_RUNG
   // the same network as SCL:
   "xv1.1" := "otw_zzaw1";
   "xv1.2" := "otw_zzaw1";
   "xv2.1" := "otw_zzaw2";
   "xv2.2" := "otw_zzaw2";
   "xv3.1" := "otw_zzaw3";
   "xv3.2" := "otw_zzaw3";
END_REGION
END_ORGANIZATION_BLOCK

ORGANIZATION_BLOCK "CyclicInterrupt"   // OB30, LAD, CyclicInterrupt
{ S7_Optimized_Access := 'TRUE' }
VERSION : 0.1
   VAR_INPUT
      Initial_Call : Bool;   // Initial call of this OB
      Event_Count : Int;   // Events discarded
   END_VAR
   VAR_TEMP
      Waga_Znormalizowana : Real;
      Rozniaca_wagi : Real;
   END_VAR
BEGIN

REGION Network 1
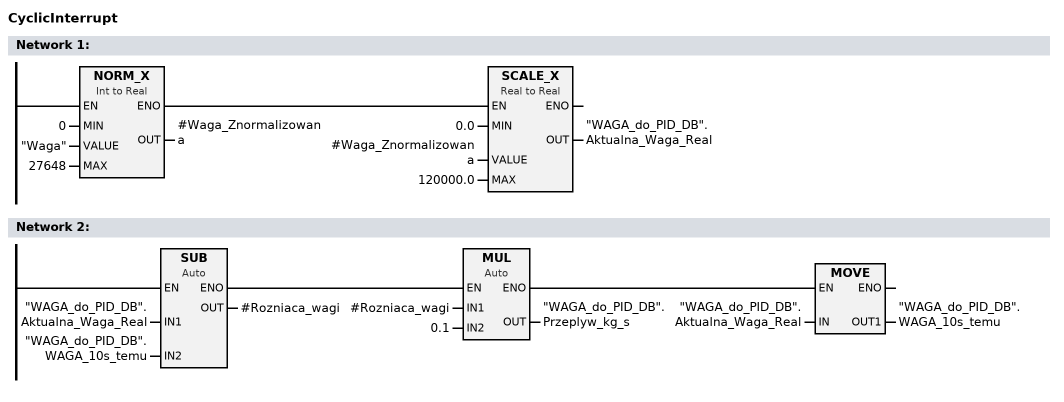
   RUNG wire#powerrail
      { S7_Templates := "[SrcType := Int, DestType := Real]" } Normalize(min := 0, value := "Waga", max := 27648, out => #Waga_Znormalizowana)
      { S7_Templates := "[SrcType := Real, DestType := Real]" } Scale(min := 0.0, value := #Waga_Znormalizowana, max := 120000.0, out => "WAGA_do_PID_DB".Aktualna_Waga_Real)
   END_RUNG
   // the same network as SCL:
   #Waga_Znormalizowana := NORM_X(MIN := 0, VALUE := "Waga", MAX := 27648);
   "WAGA_do_PID_DB".Aktualna_Waga_Real := SCALE_X(MIN := 0.0, VALUE := #Waga_Znormalizowana, MAX := 120000.0);
END_REGION

REGION Network 2
   RUNG wire#powerrail
      Sub(in1 := "WAGA_do_PID_DB".Aktualna_Waga_Real, in2 := "WAGA_do_PID_DB".WAGA_10s_temu, out => #Rozniaca_wagi)
      Mul(in1 := #Rozniaca_wagi, in2 := 0.1, out => "WAGA_do_PID_DB".Przeplyw_kg_s)
      Move(in := "WAGA_do_PID_DB".Aktualna_Waga_Real, out1 => "WAGA_do_PID_DB".WAGA_10s_temu)
   END_RUNG
   // the same network as SCL:
   #Rozniaca_wagi := "WAGA_do_PID_DB".Aktualna_Waga_Real - "WAGA_do_PID_DB".WAGA_10s_temu;
   "WAGA_do_PID_DB".Przeplyw_kg_s := #Rozniaca_wagi * 0.1;
   "WAGA_do_PID_DB".WAGA_10s_temu := "WAGA_do_PID_DB".Aktualna_Waga_Real;
END_REGION
END_ORGANIZATION_BLOCK

(* ===== HMI "HMI_RT_1" =====
system functions are stored by id; their names below are inferred from use
connection "HMI_Connection_1": ETHERNET, S7_1500_OMS

HMI tags "Default tag table"
   "lamp" : Bool = PLC M3 AT %Q8.0, 1 s
   "POT_NALEW" : Bool = PLC POT_NALEW AT %M20.7, 1 s
   "porusz_cysterne" : Bool = PLC porusz_cysterne AT %M10.1, 1 s
   "ZS_002" : Bool = PLC ZS_002 AT %I16.1, 1 s
   "ZS_001" : Bool = PLC ZS_001 AT %I16.0, 1 s
   "PROD1" : Bool = PLC PROD1 AT %M21.1, 1 s
   "Odzyskoop" : Bool = PLC Odzyskoop AT %M22.3, 1 s
   "PROD2" : Bool = PLC PROD2 AT %M21.3, 1 s
   "PROD3" : Bool = PLC PROD3 AT %M21.4, 1 s
   "STR_NALEW" : Bool = PLC STR_NALEW AT %M20.6, 1 s
   "Przycisk_Start" : Bool = PLC Przycisk_Start AT %M4.1, 1 s
   "Zrzut_paliwa" : Bool = PLC Zrzut_paliwa AT %M28.0, 1 s

HMI tags "Tag table_1"
   "HMI_Tag_1" : Int, internal
   "HMI_Tag_2" : Int, internal
   "bt1" : Bool, internal
   "bt2" : Bool, internal
   "bt3" : Bool, internal

screen "Screen_1" 1024x768
   GraphicView "Graphic view_1" at 0,596 size 521x166; Picture "Graphic_47"
      Visibility <- "porusz_cysterne"
   GraphicView "Graphic view_7" at 444,487 size 64x133; Picture "Graphic_56"
   GraphicView "Graphic view_8" at 443,317 size 65x264; Picture "Graphic_58"
   GraphicView "Graphic view_2" at 491,300 size 437x44; Picture "Graphic_71"
   GraphicView "Graphic view_3" at 453,301 size 41x42; Picture "Graphic_72"
   GraphicView "Graphic view_4" at 532,487 size 29x30; Picture "Graphic_73"
   GraphicView "Graphic view_5" at 493,490 size 43x25; Picture "Graphic_74"
   GraphicView "Graphic view_6" at 534,198 size 27x292; Picture "Graphic_75"
   GraphicView "Graphic view_9" at 530,159 size 31x46; Picture "Graphic_76"
   GraphicView "Graphic view_10" at 557,161 size 467x42; Picture "Graphic_74"
   IOField "I/O field_1" at 632,333 size 96x32; FormatPattern 9999999
   GraphicView "Graphic view_12" at 646,301 size 49x34; Picture "Graphic_78"
   IOField "I/O field_2" at 924,304 size 96x32; FormatPattern 9999999
   GraphicView "Graphic view_14" at 588,156 size 14x161; Picture "Graphic_80"
   GraphicView "Graphic view_16" at 590,133 size 11x27; Picture "Graphic_82"
   GraphicView "Graphic view_13" at 588,114 size 15x22; Picture "Graphic_84"
   Rectangle "Rectangle_5" at 602,143 size 9x9
      Appearance <- "Zrzut_paliwa"
   IOField "I/O field_3" at 110,433 size 85x26; FormatPattern 9999999
   IOField "I/O field_4" at 110,462 size 86x25; FormatPattern 9999999
   IOField "I/O field_5" at 110,490 size 86x26; FormatPattern 9999999
   Button "Button_1" at 261,309 size 159x19; TextOff 'LANCA NALEWCZA'
   Button "Button_2" at 267,336 size 146x19; TextOff 'Zezwolenie'
      Appearance <- "POT_NALEW"
   IOField "I/O field_7" at 299,515 size 42x13; FormatPattern 9999999
   IOField "I/O field_8" at 299,534 size 42x13; FormatPattern 9999999
   IOField "I/O field_9" at 299,553 size 42x13; FormatPattern 9999999
   TextField "Text field_1" at 253,514 size 17x14; Text 'Bar'
   TextField "Text field_2" at 248,534 size 45x14; Text 'Zadana_PID'
   TextField "Text field_3" at 253,553 size 35x14; Text 'Aktualna'
   GraphicView "Graphic view_15" at 23,108 size 29x25; Picture "Graphic_88"
   Button "Button_3" at 348,466 size 34x35; TextOff 'Up'
   Button "Button_4" at 388,466 size 36x35; TextOff 'DOWN'
   Button "Button_5" at 500,561 size 34x35; TextOff 'LSHH'
   TextField "Text field_4" at 53,435 size 52x20; Text 'ZADANA'
   TextField "Text field_5" at 50,465 size 60x20; Text 'Tara_min'
   TextField "Text field_6" at 47,496 size 63x20; Text 'Tara_max'
   Button "Button_6" at 379,355 size 34x35; TextOff 'LSHH'
   TextField "Text field_9" at 601,337 size 25x25; Text 'FV'
   IOField "I/O field_6" at 803,269 size 96x32; FormatPattern 9999999
   TextField "Text field_10" at 782,276 size 15x14; Text 'TT'
   GraphicView "Graphic view_18" at 535,415 size 32x54; Picture "Graphic_90"
   Rectangle "Rectangle_4" at 569,432 size 16x19
      Appearance <- "Odzyskoop"
   GraphicView "Graphic view_11" at 233,595 size 521x166; Picture "Graphic_47"
      Visibility <- "porusz_cysterne"
   Bar "Bar_2" at 282,590 size 81x139; MinimumValue 0; MaximumValue 70000
   Rectangle "Rectangle_6" at 229,729 size 24x25
      Appearance <- "ZS_001"
   TextField "Text field_11" at 232,735 size 17x14; Text 'ZS1'
   Rectangle "Rectangle_2" at 671,729 size 24x25
      Appearance <- "ZS_002"
   TextField "Text field_7" at 674,735 size 17x14; Text 'ZS2'
   Button "Button_7" at 910,362 size 96x32; TextOff 'Prod1'
      on Press: function_b14e0dd5("PROD1", 0)
      Appearance <- "PROD1"
   Button "Button_10" at 910,409 size 96x32; TextOff 'Prod2'
      on Press: function_b14e0dd5("PROD2", 0)
      Appearance <- "PROD2"
   Button "Button_11" at 910,458 size 96x32; TextOff 'Prod3'
      on Press: function_b14e0dd5("PROD3", 0)
      Appearance <- "PROD3"
   Button "Button_8" at 791,627 size 194x32; TextOff 'Start Nalewanie'
      on Press: function_b14e0dd5("STR_NALEW", 0)
   Button "Button_9" at 789,703 size 194x32; TextOff 'Start Przeciągarka'
      on Press: function_b14e0dd5("Przycisk_Start", 0)
*)